{attribute 'linkalways'}
{attribute 'no_explicit_call' := 'This FB is a CLASS and must be accessed using methods or properties'}
{attribute 'enable_dynamic_creation'}
FUNCTION_BLOCK Node_F_VN_RemapImageToPolarSpaceExp EXTENDS VisionNode
VAR
    ipSrcImage : _ITcVnImage;
    ipDestImage : _ITcVnImage;
    aCenter : _TcVnPoint2_REAL;
    fMaxRadius : _LREAL(0);
    eInterpolationType : _ETcVnInterpolationType(ETcVnInterpolationType.TCVN_IT_BILINEAR);
    hrPrev : _HRESULT(S_OK);
    hresult : _HRESULT(S_OK);
END_VAR

METHOD PUBLIC Clone : I_Node
VAR
    pNode : POINTER TO Node_F_VN_RemapImageToPolarSpaceExp;
END_VAR
pNode := __NEW(Node_F_VN_RemapImageToPolarSpaceExp);
Clone := pNode^;
END_METHOD

METHOD FB_init : BOOL
VAR_INPUT
    bInitRetains : BOOL;
    bInCopyCode : BOOL;
END_VAR
AddInput('ipSrcImage', ipSrcImage);
AddOutput('ipDestImage', ipDestImage);
AddInput('aCenter', aCenter);
AddParameter('fMaxRadius', fMaxRadius);
AddParameter('eInterpolationType', eInterpolationType);
AddInput('hrPrev', hrPrev);
AddOutput('hresult', hresult);
END_METHOD

METHOD PROTECTED OnExecute
hresult.Value := F_VN_RemapImageToPolarSpaceExp(
    ipSrcImage := ipSrcImage.Value,
    ipDestImage := ipDestImage.Value,
    aCenter := aCenter.Value,
    fMaxRadius := fMaxRadius.Value,
    eInterpolationType := eInterpolationType.Value,
    hrPrev := hrPrev.Value);
END_METHOD

METHOD PUBLIC PreExecutionCheck
VAR_INPUT
    Check : I_PreExecutionChecks;
END_VAR
Check.IsTrue(ipSrcImage.IsValid, 'ipSrcImage must contain an image');
Check.IsTrue((ipDestImage.Value = 0) OR (ipDestImage.Value <> ipSrcImage.Value), 'Destination must be different from the source image');
Check.IsTrue((eInterpolationType.Value = ETcVnInterpolationType.TCVN_IT_NEAREST_NEIGHBOR) OR
             (eInterpolationType.Value = ETcVnInterpolationType.TCVN_IT_BILINEAR) OR
             (eInterpolationType.Value = ETcVnInterpolationType.TCVN_IT_BICUBIC) OR
             (eInterpolationType.Value = ETcVnInterpolationType.TCVN_IT_AREA_BASED) OR
             (eInterpolationType.Value = ETcVnInterpolationType.TCVN_IT_LANCZOS4), 'Unsupported eInterpolationType');
Check.IsTrue(fMaxRadius.Value >= 0.0, 'Maximum radius must be non-negative; zero selects it automatically');
END_METHOD

END_FUNCTION_BLOCK

(* stored: Version 1.1.0.1, ProductVersion 3.1.4026.19
   POU Node_F_VN_RemapImageToPolarSpaceExp: Id {83e9bdba-d1f9-4544-a1a9-94a6d1204269}, SpecialFunc None
   Folder Constructor: Id {8c7e959a-b36f-479c-b3e1-700959e33e48}
   Method Clone: Id {a42938e6-f362-43b0-810b-22164e1f673f}
   Method FB_init: Id {f8b26a46-4c92-424d-aaa7-beb287041333}
   Method OnExecute: Id {8db2cc24-9c98-4765-93bb-c160ce607680}
   Method PreExecutionCheck: Id {b4debbfb-fe37-499e-bb63-ca5176d267e3} *)
